TYPE ST_RoomTempHmi :
STRUCT
	// PLC -> HMI
	nRoomTemperature		: REAL;
	sName					: STRING;
	
	// HMI -> PLC
	nValue					: INT := 5; // skaalaus HMI:ltä
	
END_STRUCT
END_TYPE

(* stored: Version 1.1.0.1
   DUT ST_RoomTempHmi: Id {f4f4a0b7-e6d2-41f2-b1fa-da251279a432} *)
